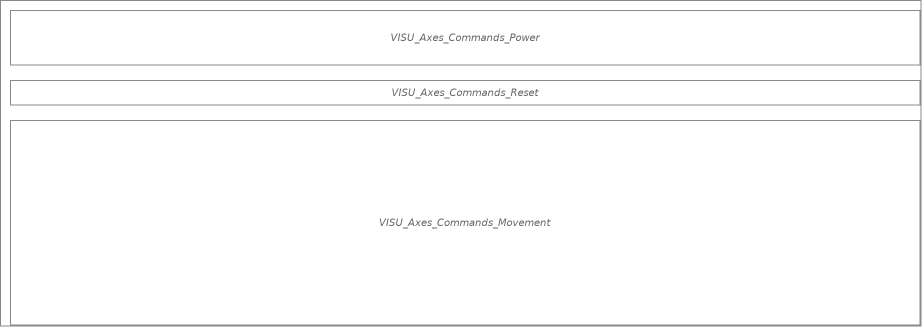
VISUALIZATION VISU_AxesRotationAxis_Processes  // 922x327
VAR_IN_OUT
	ref : AxesRotationAxis;
    ref_driveChannel : AX52XXDriveChannel;
    widget : AxesRotationAxisWidget;
END_VAR
    Frame (10,10 910x55)
        shows VISU_Axes_Commands_Power(powerOn := ref.processes.powerOn, powerOff := ref.processes.powerOff, powerOnStatus := widget.processes_powerOnStatus, powerOffStatus := widget.processes_powerOffStatus)
    Frame (10,80 910x25)
        shows VISU_Axes_Commands_Reset(reset := ref.processes.reset, resetStatus := widget.processes_resetStatus)
    Frame (10,120 910x205)
        shows VISU_Axes_Commands_Movement(stop := ref.processes.stop, moveOutOfLimitSwitch := ref.processes.moveOutOfLimitSwitch, moveAbsolute := ref.processes.moveAbsolute, moveRelative := ref.processes.moveRelative, moveVelocity := ref.processes.moveVelocity, stopStatus := widget.processes_stopStatus, moveOutOfLimitSwitchStatus := widget.processes_moveOutOfLimitSwitchStatus, moveAbsoluteStatus := widget.processes_moveAbsoluteStatus, moveRelativeStatus := widget.processes_moveRelativeStatus, moveVelocityStatus := widget.processes_moveVelocityStatus)
END_VISUALIZATION

(* stored: Version 1.1.0.1, ProductVersion 3.1.4019.2
   Visu VISU_AxesRotationAxis_Processes: Id {d1b1bd93-796c-4f82-9ec5-ab703d08871d} *)
